TYPE E_Location : (Wroclaw:=1, Warszawa, Krakow, Zakopane, Katowice, Poznan );
END_TYPE

(* stored: Version 1.1.0.1, ProductVersion 3.1.4019.2
   DUT E_Location: Id {3fba7160-fc0e-4943-bf14-601e11a27b16} *)
